Staubli VAL3: save.pgx

public program save(num& x_nResult[])
  local num i
begin
  x_nResult=saveTool:libSave()
  if x_nResult!=0
    delay(0.5)
    x_nResult=saveTool:libSave()
  endIf
end
